// TIA Portal V17 export
// export: Created 2025-03-07T09:18:44.4226865Z, ExportSetting WithDefaults, DisplayName Totally Integrated Automation Portal, DisplayVersion V17 Update 8, DisplayName TIA Portal Openness, DisplayVersion V17 Update 8, DisplayName TIA Portal Version Control Interface, DisplayVersion V17, DisplayName SINAMICS Startdrive Advanced, DisplayVersion V17 SP2, DisplayName SINAMICS Startdrive G110M, G120, G120C, G120D, G120P, G115D, DisplayVersion V17 SP2, DisplayName SINAMICS Startdrive G130, G150, S120, S150, SINAMICS MV, S210, DisplayVersion V17 SP2, DisplayName STEP 7 Professional, DisplayVersion V17 Update 8, DisplayName SINUMERIK ONE STEP 7 Toolbox, DisplayVersion V17 Update 12, DisplayName SINUMERIK 840D sl STEP 7 Toolbox, DisplayVersion V17 Update 12, DisplayName STEP 7 Safety, DisplayVersion V17 Update 6, DisplayName WinCC Advanced, DisplayVersion V17 Update 8
FUNCTION "FC2202_PROFINET" : Void   // FC2202, LAD
{ S7_Optimized_Access := 'FALSE' }
AUTHOR : ETXETAR
VERSION : 1.0
// stored: AutoNumber false, IsIECCheckEnabled false, SetENOAutomatically false, UDAEnableTagReadback false
   VAR_TEMP
      COMMAND : Int;   // COMMAND
      BUSY : Bool;   // BUSY
   END_VAR
   VAR CONSTANT
      FC_NUMBER : Int := 2202;
   END_VAR
   VAR_TEMP   // added for the SCL form of the ladder/FBD networks
      _w1 : Bool;
   END_VAR
BEGIN

REGION Network 1: PROFINET HMI COMMUNICATION
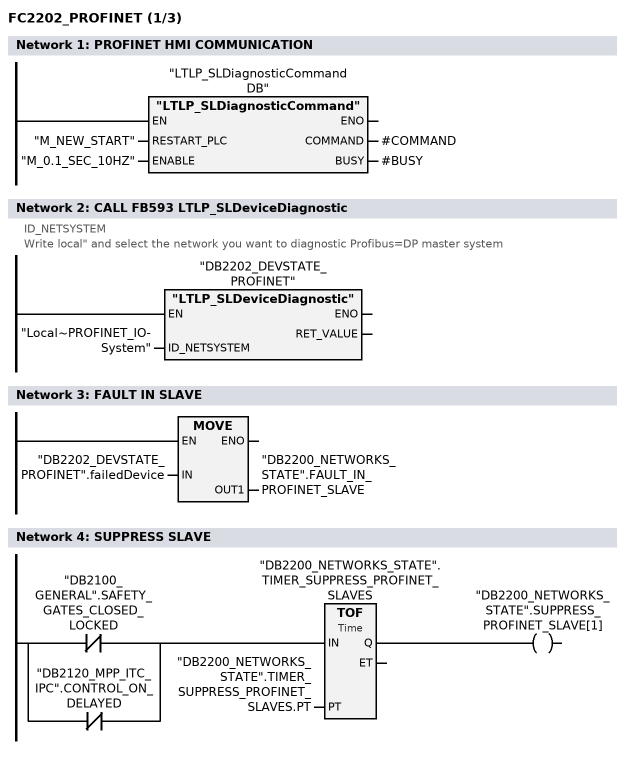
   RUNG wire#powerrail
      "LTLP_SLDiagnosticCommandDB"(RESTART_PLC := "M_NEW_START", ENABLE := "M_0.1_SEC_10HZ", COMMAND => #COMMAND, BUSY => #BUSY)
   END_RUNG
   // the same network as SCL:
   "LTLP_SLDiagnosticCommandDB"(RESTART_PLC := "M_NEW_START",   // "LTLP_SLDiagnosticCommand"
                           ENABLE := "M_0.1_SEC_10HZ",
                           COMMAND => #COMMAND,
                           BUSY => #BUSY);
END_REGION

REGION Network 2: CALL FB593 LTLP_SLDeviceDiagnostic
   // ID_NETSYSTEM
   // Write local" and select the network you want to diagnostic Profibus=DP master system
   RUNG wire#powerrail
      "DB2202_DEVSTATE_PROFINET"(ID_NETSYSTEM := "Local~PROFINET_IO-System", RET_VALUE =>)
   END_RUNG
   // the same network as SCL:
   "DB2202_DEVSTATE_PROFINET"(ID_NETSYSTEM := "Local~PROFINET_IO-System");   // "LTLP_SLDeviceDiagnostic"
END_REGION

REGION Network 3: FAULT IN SLAVE
   RUNG wire#powerrail
      Move(in := "DB2202_DEVSTATE_PROFINET".failedDevice, out1 => "DB2200_NETWORKS_STATE".FAULT_IN_PROFINET_SLAVE)
   END_RUNG
   // the same network as SCL:
   "DB2200_NETWORKS_STATE".FAULT_IN_PROFINET_SLAVE := "DB2202_DEVSTATE_PROFINET".failedDevice;
END_REGION

REGION Network 4: SUPPRESS SLAVE
   RUNG wire#powerrail
      I_Contact( "DB2100_GENERAL".SAFETY_GATES_CLOSED_LOCKED )
      wire#w1
      { S7_Templates := "time_type := Time" } "DB2200_NETWORKS_STATE".TIMER_SUPPRESS_PROFINET_SLAVES.TOF(pt := "DB2200_NETWORKS_STATE".TIMER_SUPPRESS_PROFINET_SLAVES.PT, et =>)
      Coil( "DB2200_NETWORKS_STATE".SUPPRESS_PROFINET_SLAVE[1] )
   END_RUNG
   RUNG wire#powerrail
      I_Contact( "DB2120_MPP_ITC_IPC".CONTROL_ON_DELAYED )
   END_RUNG wire#w1
   // the same network as SCL:
   "DB2200_NETWORKS_STATE".TIMER_SUPPRESS_PROFINET_SLAVES.TOF(IN := NOT "DB2100_GENERAL".SAFETY_GATES_CLOSED_LOCKED OR NOT "DB2120_MPP_ITC_IPC".CONTROL_ON_DELAYED,
                           PT := "DB2200_NETWORKS_STATE".TIMER_SUPPRESS_PROFINET_SLAVES.PT);
   "DB2200_NETWORKS_STATE".SUPPRESS_PROFINET_SLAVE[1] := "DB2200_NETWORKS_STATE".TIMER_SUPPRESS_PROFINET_SLAVES.Q;
END_REGION

REGION Network 5: PROFINET IMMEDIATE STOP ALARMS
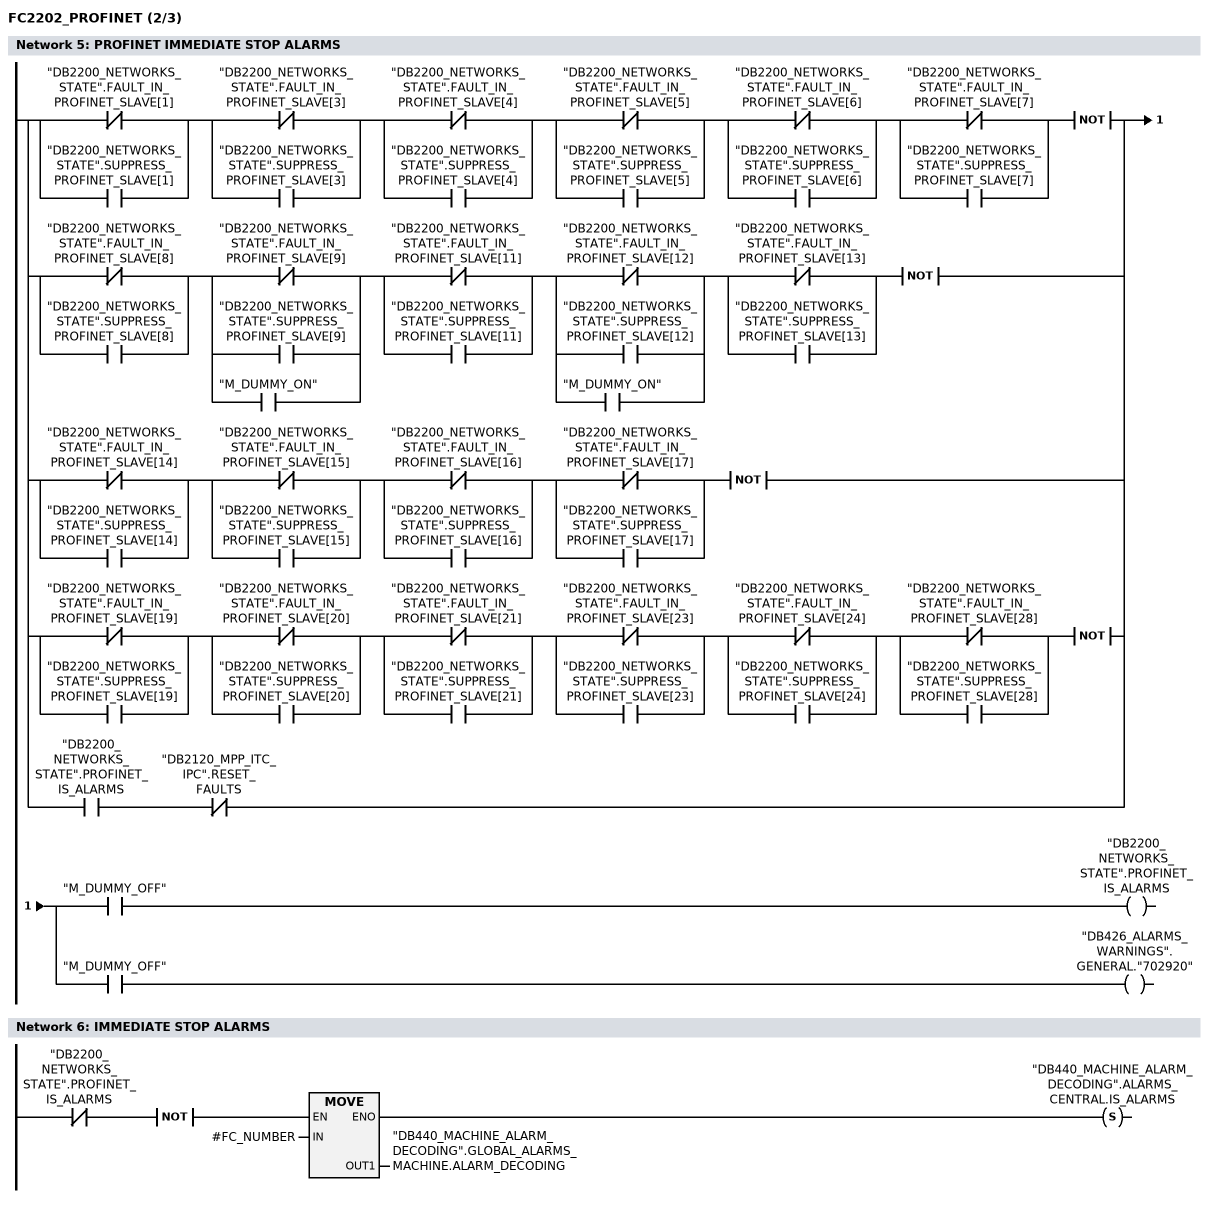
   RUNG wire#powerrail
      I_Contact( "DB2200_NETWORKS_STATE".FAULT_IN_PROFINET_SLAVE[1] )
      wire#w1
      I_Contact( "DB2200_NETWORKS_STATE".FAULT_IN_PROFINET_SLAVE[3] )
      wire#w2
      I_Contact( "DB2200_NETWORKS_STATE".FAULT_IN_PROFINET_SLAVE[4] )
      wire#w3
      I_Contact( "DB2200_NETWORKS_STATE".FAULT_IN_PROFINET_SLAVE[5] )
      wire#w4
      I_Contact( "DB2200_NETWORKS_STATE".FAULT_IN_PROFINET_SLAVE[6] )
      wire#w5
      I_Contact( "DB2200_NETWORKS_STATE".FAULT_IN_PROFINET_SLAVE[7] )
      wire#w6
      Not()
      wire#w7
      Contact( "M_DUMMY_OFF" )
      Coil( "DB2200_NETWORKS_STATE".PROFINET_IS_ALARMS )
   END_RUNG
   RUNG wire#powerrail
      Contact( "DB2200_NETWORKS_STATE".SUPPRESS_PROFINET_SLAVE[1] )
   END_RUNG wire#w1
   RUNG wire#w1
      Contact( "DB2200_NETWORKS_STATE".SUPPRESS_PROFINET_SLAVE[3] )
   END_RUNG wire#w2
   RUNG wire#w2
      Contact( "DB2200_NETWORKS_STATE".SUPPRESS_PROFINET_SLAVE[4] )
   END_RUNG wire#w3
   RUNG wire#w3
      Contact( "DB2200_NETWORKS_STATE".SUPPRESS_PROFINET_SLAVE[5] )
   END_RUNG wire#w4
   RUNG wire#w4
      Contact( "DB2200_NETWORKS_STATE".SUPPRESS_PROFINET_SLAVE[6] )
   END_RUNG wire#w5
   RUNG wire#w5
      Contact( "DB2200_NETWORKS_STATE".SUPPRESS_PROFINET_SLAVE[7] )
   END_RUNG wire#w6
   RUNG wire#powerrail
      I_Contact( "DB2200_NETWORKS_STATE".FAULT_IN_PROFINET_SLAVE[8] )
      wire#w8
      I_Contact( "DB2200_NETWORKS_STATE".FAULT_IN_PROFINET_SLAVE[9] )
      wire#w9
      I_Contact( "DB2200_NETWORKS_STATE".FAULT_IN_PROFINET_SLAVE[11] )
      wire#w10
      I_Contact( "DB2200_NETWORKS_STATE".FAULT_IN_PROFINET_SLAVE[12] )
      wire#w11
      I_Contact( "DB2200_NETWORKS_STATE".FAULT_IN_PROFINET_SLAVE[13] )
      wire#w12
      Not()
   END_RUNG wire#w7
   RUNG wire#powerrail
      Contact( "DB2200_NETWORKS_STATE".SUPPRESS_PROFINET_SLAVE[8] )
   END_RUNG wire#w8
   RUNG wire#w8
      Contact( "DB2200_NETWORKS_STATE".SUPPRESS_PROFINET_SLAVE[9] )
   END_RUNG wire#w9
   RUNG wire#w8
      Contact( "M_DUMMY_ON" )
   END_RUNG wire#w9
   RUNG wire#w9
      Contact( "DB2200_NETWORKS_STATE".SUPPRESS_PROFINET_SLAVE[11] )
   END_RUNG wire#w10
   RUNG wire#w10
      Contact( "DB2200_NETWORKS_STATE".SUPPRESS_PROFINET_SLAVE[12] )
   END_RUNG wire#w11
   RUNG wire#w10
      Contact( "M_DUMMY_ON" )
   END_RUNG wire#w11
   RUNG wire#w11
      Contact( "DB2200_NETWORKS_STATE".SUPPRESS_PROFINET_SLAVE[13] )
   END_RUNG wire#w12
   RUNG wire#powerrail
      I_Contact( "DB2200_NETWORKS_STATE".FAULT_IN_PROFINET_SLAVE[14] )
      wire#w13
      I_Contact( "DB2200_NETWORKS_STATE".FAULT_IN_PROFINET_SLAVE[15] )
      wire#w14
      I_Contact( "DB2200_NETWORKS_STATE".FAULT_IN_PROFINET_SLAVE[16] )
      wire#w15
      I_Contact( "DB2200_NETWORKS_STATE".FAULT_IN_PROFINET_SLAVE[17] )
      wire#w16
      Not()
   END_RUNG wire#w7
   RUNG wire#powerrail
      Contact( "DB2200_NETWORKS_STATE".SUPPRESS_PROFINET_SLAVE[14] )
   END_RUNG wire#w13
   RUNG wire#w13
      Contact( "DB2200_NETWORKS_STATE".SUPPRESS_PROFINET_SLAVE[15] )
   END_RUNG wire#w14
   RUNG wire#w14
      Contact( "DB2200_NETWORKS_STATE".SUPPRESS_PROFINET_SLAVE[16] )
   END_RUNG wire#w15
   RUNG wire#w15
      Contact( "DB2200_NETWORKS_STATE".SUPPRESS_PROFINET_SLAVE[17] )
   END_RUNG wire#w16
   RUNG wire#powerrail
      I_Contact( "DB2200_NETWORKS_STATE".FAULT_IN_PROFINET_SLAVE[19] )
      wire#w17
      I_Contact( "DB2200_NETWORKS_STATE".FAULT_IN_PROFINET_SLAVE[20] )
      wire#w18
      I_Contact( "DB2200_NETWORKS_STATE".FAULT_IN_PROFINET_SLAVE[21] )
      wire#w19
      I_Contact( "DB2200_NETWORKS_STATE".FAULT_IN_PROFINET_SLAVE[23] )
      wire#w20
      I_Contact( "DB2200_NETWORKS_STATE".FAULT_IN_PROFINET_SLAVE[24] )
      wire#w21
      I_Contact( "DB2200_NETWORKS_STATE".FAULT_IN_PROFINET_SLAVE[28] )
      wire#w22
      Not()
   END_RUNG wire#w7
   RUNG wire#powerrail
      Contact( "DB2200_NETWORKS_STATE".SUPPRESS_PROFINET_SLAVE[19] )
   END_RUNG wire#w17
   RUNG wire#w17
      Contact( "DB2200_NETWORKS_STATE".SUPPRESS_PROFINET_SLAVE[20] )
   END_RUNG wire#w18
   RUNG wire#w18
      Contact( "DB2200_NETWORKS_STATE".SUPPRESS_PROFINET_SLAVE[21] )
   END_RUNG wire#w19
   RUNG wire#w19
      Contact( "DB2200_NETWORKS_STATE".SUPPRESS_PROFINET_SLAVE[23] )
   END_RUNG wire#w20
   RUNG wire#w20
      Contact( "DB2200_NETWORKS_STATE".SUPPRESS_PROFINET_SLAVE[24] )
   END_RUNG wire#w21
   RUNG wire#w21
      Contact( "DB2200_NETWORKS_STATE".SUPPRESS_PROFINET_SLAVE[28] )
   END_RUNG wire#w22
   RUNG wire#powerrail
      Contact( "DB2200_NETWORKS_STATE".PROFINET_IS_ALARMS )
      I_Contact( "DB2120_MPP_ITC_IPC".RESET_FAULTS )
   END_RUNG wire#w7
   RUNG wire#w7
      Contact( "M_DUMMY_OFF" )
      Coil( "DB426_ALARMS_WARNINGS".GENERAL."702920" )
   END_RUNG
   // the same network as SCL:
   #_w1 := NOT ((NOT "DB2200_NETWORKS_STATE".FAULT_IN_PROFINET_SLAVE[1] OR "DB2200_NETWORKS_STATE".SUPPRESS_PROFINET_SLAVE[1]) AND (NOT "DB2200_NETWORKS_STATE".FAULT_IN_PROFINET_SLAVE[3] OR "DB2200_NETWORKS_STATE".SUPPRESS_PROFINET_SLAVE[3]) AND (NOT "DB2200_NETWORKS_STATE".FAULT_IN_PROFINET_SLAVE[4] OR "DB2200_NETWORKS_STATE".SUPPRESS_PROFINET_SLAVE[4]) AND (NOT "DB2200_NETWORKS_STATE".FAULT_IN_PROFINET_SLAVE[5] OR "DB2200_NETWORKS_STATE".SUPPRESS_PROFINET_SLAVE[5]) AND (NOT "DB2200_NETWORKS_STATE".FAULT_IN_PROFINET_SLAVE[6] OR "DB2200_NETWORKS_STATE".SUPPRESS_PROFINET_SLAVE[6]) AND (NOT "DB2200_NETWORKS_STATE".FAULT_IN_PROFINET_SLAVE[7] OR "DB2200_NETWORKS_STATE".SUPPRESS_PROFINET_SLAVE[7])) OR NOT ((NOT "DB2200_NETWORKS_STATE".FAULT_IN_PROFINET_SLAVE[8] OR "DB2200_NETWORKS_STATE".SUPPRESS_PROFINET_SLAVE[8]) AND (NOT "DB2200_NETWORKS_STATE".FAULT_IN_PROFINET_SLAVE[9] OR "DB2200_NETWORKS_STATE".SUPPRESS_PROFINET_SLAVE[9] OR "M_DUMMY_ON") AND (NOT "DB2200_NETWORKS_STATE".FAULT_IN_PROFINET_SLAVE[11] OR "DB2200_NETWORKS_STATE".SUPPRESS_PROFINET_SLAVE[11]) AND (NOT "DB2200_NETWORKS_STATE".FAULT_IN_PROFINET_SLAVE[12] OR "DB2200_NETWORKS_STATE".SUPPRESS_PROFINET_SLAVE[12] OR "M_DUMMY_ON") AND (NOT "DB2200_NETWORKS_STATE".FAULT_IN_PROFINET_SLAVE[13] OR "DB2200_NETWORKS_STATE".SUPPRESS_PROFINET_SLAVE[13])) OR NOT ((NOT "DB2200_NETWORKS_STATE".FAULT_IN_PROFINET_SLAVE[14] OR "DB2200_NETWORKS_STATE".SUPPRESS_PROFINET_SLAVE[14]) AND (NOT "DB2200_NETWORKS_STATE".FAULT_IN_PROFINET_SLAVE[15] OR "DB2200_NETWORKS_STATE".SUPPRESS_PROFINET_SLAVE[15]) AND (NOT "DB2200_NETWORKS_STATE".FAULT_IN_PROFINET_SLAVE[16] OR "DB2200_NETWORKS_STATE".SUPPRESS_PROFINET_SLAVE[16]) AND (NOT "DB2200_NETWORKS_STATE".FAULT_IN_PROFINET_SLAVE[17] OR "DB2200_NETWORKS_STATE".SUPPRESS_PROFINET_SLAVE[17])) OR NOT ((NOT "DB2200_NETWORKS_STATE".FAULT_IN_PROFINET_SLAVE[19] OR "DB2200_NETWORKS_STATE".SUPPRESS_PROFINET_SLAVE[19]) AND (NOT "DB2200_NETWORKS_STATE".FAULT_IN_PROFINET_SLAVE[20] OR "DB2200_NETWORKS_STATE".SUPPRESS_PROFINET_SLAVE[20]) AND (NOT "DB2200_NETWORKS_STATE".FAULT_IN_PROFINET_SLAVE[21] OR "DB2200_NETWORKS_STATE".SUPPRESS_PROFINET_SLAVE[21]) AND (NOT "DB2200_NETWORKS_STATE".FAULT_IN_PROFINET_SLAVE[23] OR "DB2200_NETWORKS_STATE".SUPPRESS_PROFINET_SLAVE[23]) AND (NOT "DB2200_NETWORKS_STATE".FAULT_IN_PROFINET_SLAVE[24] OR "DB2200_NETWORKS_STATE".SUPPRESS_PROFINET_SLAVE[24]) AND (NOT "DB2200_NETWORKS_STATE".FAULT_IN_PROFINET_SLAVE[28] OR "DB2200_NETWORKS_STATE".SUPPRESS_PROFINET_SLAVE[28])) OR ("DB2200_NETWORKS_STATE".PROFINET_IS_ALARMS AND NOT "DB2120_MPP_ITC_IPC".RESET_FAULTS);
   "DB2200_NETWORKS_STATE".PROFINET_IS_ALARMS := #_w1 AND "M_DUMMY_OFF";
   "DB426_ALARMS_WARNINGS".GENERAL."702920" := #_w1 AND "M_DUMMY_OFF";
END_REGION

REGION Network 6: IMMEDIATE STOP ALARMS
   RUNG wire#powerrail
      I_Contact( "DB2200_NETWORKS_STATE".PROFINET_IS_ALARMS )
      Not()
      { S7_GenerateENO := "TRUE" } Move(in := #FC_NUMBER, out1 => "DB440_MACHINE_ALARM_DECODING".GLOBAL_ALARMS_MACHINE.ALARM_DECODING)
      S_Coil( "DB440_MACHINE_ALARM_DECODING".ALARMS_CENTRAL.IS_ALARMS )
   END_RUNG
   // the same network as SCL:
   // ENO of a box is taken as its EN; it also drops when the box reports an error
   IF NOT (NOT "DB2200_NETWORKS_STATE".PROFINET_IS_ALARMS) THEN
       "DB440_MACHINE_ALARM_DECODING".GLOBAL_ALARMS_MACHINE.ALARM_DECODING := #FC_NUMBER;
       "DB440_MACHINE_ALARM_DECODING".ALARMS_CENTRAL.IS_ALARMS := TRUE;
   END_IF;
END_REGION

REGION Network 7: PROFINET STOP END OF CYCLE ALARMS
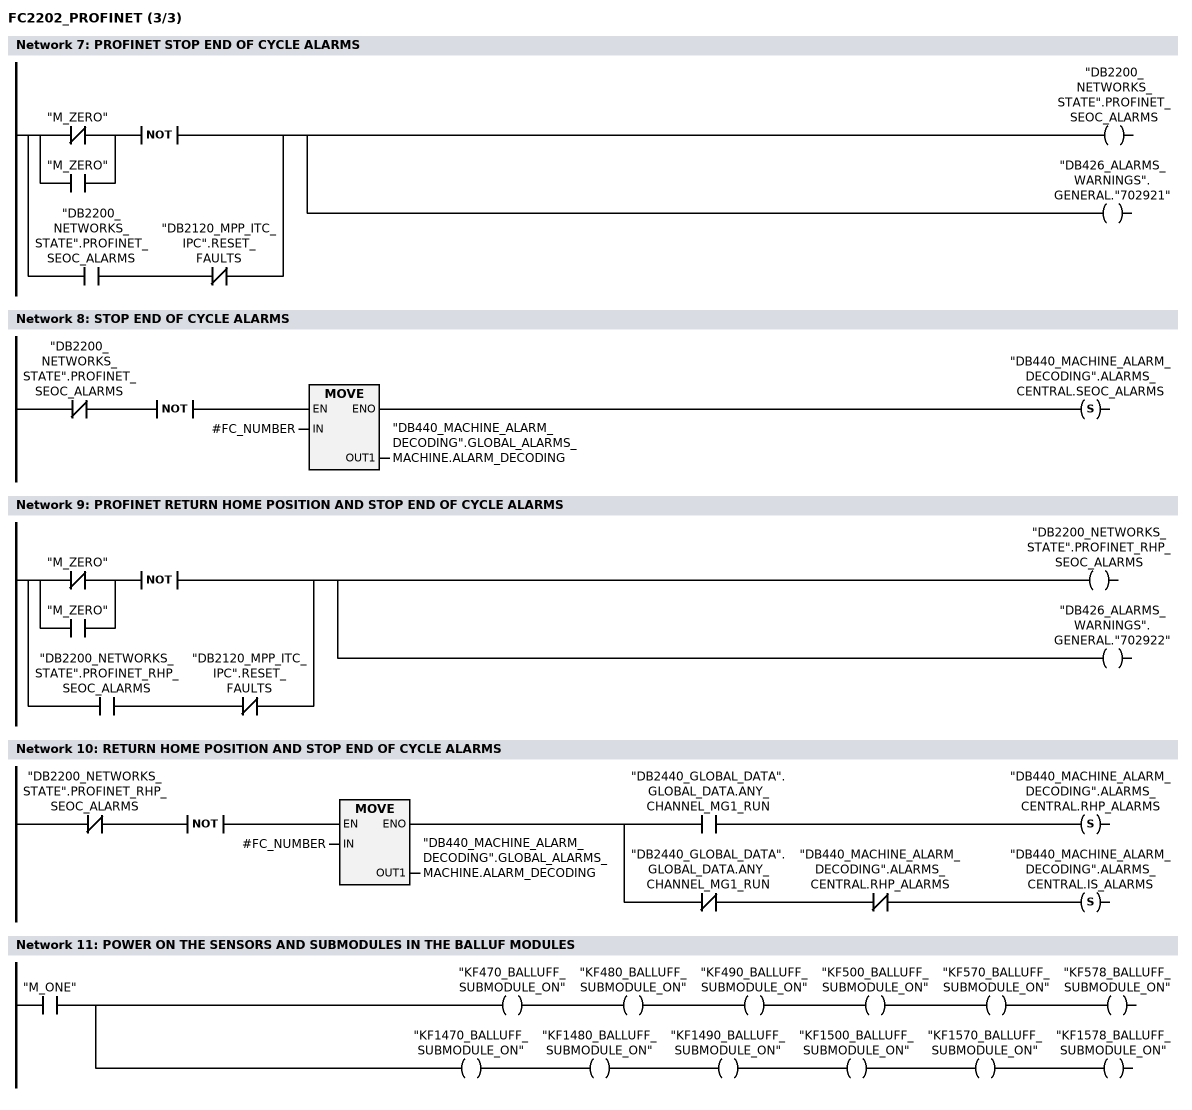
   RUNG wire#powerrail
      I_Contact( "M_ZERO" )
      wire#w1
      Not()
      wire#w2
      Coil( "DB2200_NETWORKS_STATE".PROFINET_SEOC_ALARMS )
   END_RUNG
   RUNG wire#powerrail
      Contact( "M_ZERO" )
   END_RUNG wire#w1
   RUNG wire#powerrail
      Contact( "DB2200_NETWORKS_STATE".PROFINET_SEOC_ALARMS )
      I_Contact( "DB2120_MPP_ITC_IPC".RESET_FAULTS )
   END_RUNG wire#w2
   RUNG wire#w2
      Coil( "DB426_ALARMS_WARNINGS".GENERAL."702921" )
   END_RUNG
   // the same network as SCL:
   "DB2200_NETWORKS_STATE".PROFINET_SEOC_ALARMS := NOT (NOT "M_ZERO" OR "M_ZERO") OR ("DB2200_NETWORKS_STATE".PROFINET_SEOC_ALARMS AND NOT "DB2120_MPP_ITC_IPC".RESET_FAULTS);
   "DB426_ALARMS_WARNINGS".GENERAL."702921" := "DB2200_NETWORKS_STATE".PROFINET_SEOC_ALARMS;
END_REGION

REGION Network 8: STOP END OF CYCLE ALARMS
   RUNG wire#powerrail
      I_Contact( "DB2200_NETWORKS_STATE".PROFINET_SEOC_ALARMS )
      Not()
      { S7_GenerateENO := "TRUE" } Move(in := #FC_NUMBER, out1 => "DB440_MACHINE_ALARM_DECODING".GLOBAL_ALARMS_MACHINE.ALARM_DECODING)
      S_Coil( "DB440_MACHINE_ALARM_DECODING".ALARMS_CENTRAL.SEOC_ALARMS )
   END_RUNG
   // the same network as SCL:
   // ENO of a box is taken as its EN; it also drops when the box reports an error
   IF NOT (NOT "DB2200_NETWORKS_STATE".PROFINET_SEOC_ALARMS) THEN
       "DB440_MACHINE_ALARM_DECODING".GLOBAL_ALARMS_MACHINE.ALARM_DECODING := #FC_NUMBER;
       "DB440_MACHINE_ALARM_DECODING".ALARMS_CENTRAL.SEOC_ALARMS := TRUE;
   END_IF;
END_REGION

REGION Network 9: PROFINET RETURN HOME POSITION AND STOP END OF CYCLE ALARMS
   RUNG wire#powerrail
      I_Contact( "M_ZERO" )
      wire#w1
      Not()
      wire#w2
      Coil( "DB2200_NETWORKS_STATE".PROFINET_RHP_SEOC_ALARMS )
   END_RUNG
   RUNG wire#powerrail
      Contact( "M_ZERO" )
   END_RUNG wire#w1
   RUNG wire#powerrail
      Contact( "DB2200_NETWORKS_STATE".PROFINET_RHP_SEOC_ALARMS )
      I_Contact( "DB2120_MPP_ITC_IPC".RESET_FAULTS )
   END_RUNG wire#w2
   RUNG wire#w2
      Coil( "DB426_ALARMS_WARNINGS".GENERAL."702922" )
   END_RUNG
   // the same network as SCL:
   "DB2200_NETWORKS_STATE".PROFINET_RHP_SEOC_ALARMS := NOT (NOT "M_ZERO" OR "M_ZERO") OR ("DB2200_NETWORKS_STATE".PROFINET_RHP_SEOC_ALARMS AND NOT "DB2120_MPP_ITC_IPC".RESET_FAULTS);
   "DB426_ALARMS_WARNINGS".GENERAL."702922" := "DB2200_NETWORKS_STATE".PROFINET_RHP_SEOC_ALARMS;
END_REGION

REGION Network 10: RETURN HOME POSITION AND STOP END OF CYCLE ALARMS
   RUNG wire#powerrail
      I_Contact( "DB2200_NETWORKS_STATE".PROFINET_RHP_SEOC_ALARMS )
      Not()
      { S7_GenerateENO := "TRUE" } Move(in := #FC_NUMBER, out1 => "DB440_MACHINE_ALARM_DECODING".GLOBAL_ALARMS_MACHINE.ALARM_DECODING)
      wire#w1
      Contact( "DB2440_GLOBAL_DATA".GLOBAL_DATA.ANY_CHANNEL_MG1_RUN )
      S_Coil( "DB440_MACHINE_ALARM_DECODING".ALARMS_CENTRAL.RHP_ALARMS )
   END_RUNG
   RUNG wire#w1
      I_Contact( "DB2440_GLOBAL_DATA".GLOBAL_DATA.ANY_CHANNEL_MG1_RUN )
      I_Contact( "DB440_MACHINE_ALARM_DECODING".ALARMS_CENTRAL.RHP_ALARMS )
      S_Coil( "DB440_MACHINE_ALARM_DECODING".ALARMS_CENTRAL.IS_ALARMS )
   END_RUNG
   // the same network as SCL:
   // ENO of a box is taken as its EN; it also drops when the box reports an error
   #_w1 := NOT (NOT "DB2200_NETWORKS_STATE".PROFINET_RHP_SEOC_ALARMS);
   IF #_w1 THEN "DB440_MACHINE_ALARM_DECODING".GLOBAL_ALARMS_MACHINE.ALARM_DECODING := #FC_NUMBER; END_IF;
   IF #_w1 AND "DB2440_GLOBAL_DATA".GLOBAL_DATA.ANY_CHANNEL_MG1_RUN THEN
       "DB440_MACHINE_ALARM_DECODING".ALARMS_CENTRAL.RHP_ALARMS := TRUE;
   END_IF;
   IF #_w1 AND NOT "DB2440_GLOBAL_DATA".GLOBAL_DATA.ANY_CHANNEL_MG1_RUN AND NOT "DB440_MACHINE_ALARM_DECODING".ALARMS_CENTRAL.RHP_ALARMS THEN
       "DB440_MACHINE_ALARM_DECODING".ALARMS_CENTRAL.IS_ALARMS := TRUE;
   END_IF;
END_REGION

REGION Network 11: POWER ON THE SENSORS AND SUBMODULES IN THE BALLUF MODULES
   RUNG wire#powerrail
      Contact( "M_ONE" )
      wire#w1
      Coil( "KF470_BALLUFF_SUBMODULE_ON" )
      Coil( "KF480_BALLUFF_SUBMODULE_ON" )
      Coil( "KF490_BALLUFF_SUBMODULE_ON" )
      Coil( "KF500_BALLUFF_SUBMODULE_ON" )
      Coil( "KF570_BALLUFF_SUBMODULE_ON" )
      Coil( "KF578_BALLUFF_SUBMODULE_ON" )
   END_RUNG
   RUNG wire#w1
      Coil( "KF1470_BALLUFF_SUBMODULE_ON" )
      Coil( "KF1480_BALLUFF_SUBMODULE_ON" )
      Coil( "KF1490_BALLUFF_SUBMODULE_ON" )
      Coil( "KF1500_BALLUFF_SUBMODULE_ON" )
      Coil( "KF1570_BALLUFF_SUBMODULE_ON" )
      Coil( "KF1578_BALLUFF_SUBMODULE_ON" )
   END_RUNG
   // the same network as SCL:
   "KF470_BALLUFF_SUBMODULE_ON" := "M_ONE";
   "KF480_BALLUFF_SUBMODULE_ON" := "M_ONE";
   "KF490_BALLUFF_SUBMODULE_ON" := "M_ONE";
   "KF500_BALLUFF_SUBMODULE_ON" := "M_ONE";
   "KF570_BALLUFF_SUBMODULE_ON" := "M_ONE";
   "KF578_BALLUFF_SUBMODULE_ON" := "M_ONE";
   "KF1470_BALLUFF_SUBMODULE_ON" := "M_ONE";
   "KF1480_BALLUFF_SUBMODULE_ON" := "M_ONE";
   "KF1490_BALLUFF_SUBMODULE_ON" := "M_ONE";
   "KF1500_BALLUFF_SUBMODULE_ON" := "M_ONE";
   "KF1570_BALLUFF_SUBMODULE_ON" := "M_ONE";
   "KF1578_BALLUFF_SUBMODULE_ON" := "M_ONE";
END_REGION
END_FUNCTION
